TYPE MyStructure :
STRUCT
    member1     : LREAL; // Some member
END_STRUCT
END_TYPE

(* stored: Version 1.1.0.1, ProductVersion 3.1.4024.11
   DUT MyStructure: Id {8d544980-d09e-407f-a9cb-828de0e99a90} *)
